# EPICS StreamDevice protocol: riesling/riesling22/device_config/riesling22.proto
Terminator = LF;

getVersion {
	out "v";
	in "v %#s";
}

getCurrent {
	in ">%e";
}

setRange {
	out "r%{0|1}";
	in "r%{0|1}";
	@init {
		out "r";
		in "r%{0|1}";
	}
}

getRange {
	in "r%{0|1}";
}

setAutoRange {
	out "u%{0|1}";
	in "u%{0|1}";
	@init {
		out "u";
		in "u%{0|1}";
	}
}

setEnable {
	out "e%{0|1}";
	in "e%{0|1}";
	@init {
		out "e";
		in "e%{0|1}";
	}
}

getEnable {
	in "e%{0|1}";
}

setAveraging {
	out "a%d";
	in "a%d";
	@init {
		out "a";
		in "a%d";
	}
}
